FUNCTION_BLOCK CylControlILAdpOL (* Composite Function Block Type *)
  (* Standard: 61499-2 *)
  (* Version 0.0, 7/14/2023, valeriy, nxtControl GmBH, template *)
  PACKAGE Main;
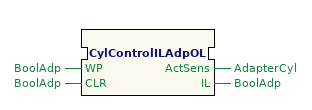
  SOCKETS
    WP : BoolAdp;
    CLR : BoolAdp;
  END_SOCKETS
  PLUGS
    ActSens : AdapterCyl;
    IL : BoolAdp;
  END_PLUGS
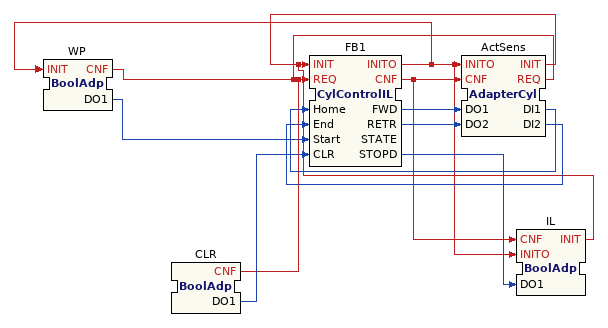
  FBS
    FB1 : CylControlIL;
  END_FBS
  EVENT_CONNECTIONS
    FB1.INITO TO ActSens.INITO;
    FB1.CNF TO ActSens.CNF;
    FB1.INITO TO WP.INIT;
    WP.CNF TO FB1.REQ;
    ActSens.INIT TO FB1.INIT;
    CLR.CNF TO FB1.REQ;
    FB1.CNF TO IL.CNF;
    FB1.INITO TO IL.INITO;
    IL.INIT TO FB1.INIT;
    ActSens.REQ TO FB1.REQ;
  END_CONNECTIONS
  DATA_CONNECTIONS
    WP.DO1 TO FB1.Start;
    FB1.STOPD TO IL.DO1;
    ActSens.DI1 TO FB1.Home;
    ActSens.DI2 TO FB1.End;
    FB1.FWD TO ActSens.DO1;
    FB1.RETR TO ActSens.DO2;
    CLR.DO1 TO FB1.CLR;
  END_CONNECTIONS
END_FUNCTION_BLOCK
